TYPE IO_In_Typ :
STRUCT
	PrimeryPressFeedback :fb_io_in_bool;
	SeconderyPressFeedbak:fb_io_in_bool;
	E_StopPressed  	: BOOL;
	E_StopPressedRaw AT %I* 	: BOOL;
	
	UW_1_Diameter AT %I* 	: INT;
	UW_2_Diameter AT %I* 	: INT;
	UW_1_LoacCell AT %I* 	: DINT;
	UW_2_LoacCell AT %I* 	: DINT;	
	
	UW_1_DancerFull AT %I* 	: BOOL;
	UW_2_DancerFull AT %I* 	: BOOL;
	
	UW_1_DancerPosition AT %I* 	: INT;
	UW_2_DancerPosition AT %I* 	: INT;

	HomeOutAxis	 AT %I* 	: BOOL;
	
	
END_STRUCT
END_TYPE

(* stored: Version 1.1.0.1, ProductVersion 3.1.4024.3
   DUT IO_In_Typ: Id {d9092035-590a-4ea9-8869-60aa4efc0d42} *)
